// TIA Portal V16 export
// export: Created 2021-05-31T23:53:35.7310699Z, ExportSetting WithDefaults, DisplayName Totally Integrated Automation Portal, DisplayVersion V16 Update 4, DisplayName TIA Portal Version Control Interface, DisplayVersion V16 Update 2, DisplayName TIA Portal Openness, DisplayVersion V16 Update 4, DisplayName STEP 7 Professional, DisplayVersion V16 Update 4, DisplayName STEP 7 Safety, DisplayVersion V16, DisplayName WinCC Advanced, DisplayVersion V16 Update 4
FUNCTION "UserAnd" : Void   // FC1, F_FBD
{ S7_Optimized_Access := 'TRUE' }
VERSION : 0.1
// stored: AutoNumber true, IsIECCheckEnabled false, UDAEnableTagReadback false
   VAR_INPUT
      "a" : Bool;
      "b" : Bool;
   END_VAR
   VAR_OUTPUT
      a_and_b : Bool;
   END_VAR
BEGIN

REGION Network 1
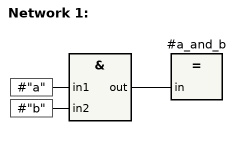
   #a_and_b := #"a" AND #"b";
END_REGION
END_FUNCTION
